PROGRAM MAIN
VAR
END_VAR

END_PROGRAM

(* stored: Version 1.1.0.1
   POU MAIN: Id {0377af76-11f4-4039-a583-64fa3f16a6eb} *)
